PROGRAM P93_Setting
VAR

	
END_VAR

END_PROGRAM

(* stored: Version 1.1.0.1, ProductVersion 3.1.4024.12
   POU P93_Setting: Id {291d468a-e342-4faf-8035-4ed6f7eda84b}, SpecialFunc None *)
